// [Sample]
// User specific weather station.
FUNCTION_BLOCK FB_BA_MyWeatherStation EXTENDS FB_BA_Publisher IMPLEMENTS I_BA_MyWeatherStation
VAR_OUTPUT
	fWeatherTemperature	: REAL;
	fHumidity			: REAL;
	fBrightness			: REAL;
	
	bDisturb			: BOOL;
END_VAR
VAR
	{region 'Internal'}
		eState			: (eInit:=1, eOperation:=2, eError:=3) UDINT	:= 1;
		stData			: ST_BA_MyWeatherData;
	{endregion}
	{region 'Temporary'}
		_nCounter		: UINT;
	{endregion}
END_VAR

CASE (eState) OF
	eInit:
		IF (OnInit()) THEN
			eState := eOperation;
		ELSE
			eState := eError;
		END_IF
		
	eOperation:
		// [Sample] Simulate weather data.
		_nCounter := (_nCounter+1);
		
		IF ((_nCounter MOD 1000) > 800) THEN
			// Simulate a physical error:
			MEMSET(ADR(stData), 0, SIZEOF(stData));
			stData.fWeatherTemperature := 99.9;
			stData.fHumidity := 99.9;
			stData.bDisturb := TRUE;
		ELSE
			// Simulate valid values:
			stData.fWeatherTemperature := 20 + (TO_REAL((_nCounter / 10) MOD 100) * 0.01);
			stData.fHumidity := TO_REAL(50 + (_nCounter MOD 1000) / 500);
			stData.fBrightness := TO_REAL(10 + (_nCounter MOD 1000) / 200);
			stData.fWindSpeed := TO_REAL(5 + ((_nCounter MOD 500) / 10));
			stData.fWindDirection := TO_REAL(90 + ((_nCounter MOD 500) / 200));
			stData.fLatitude := 51.8761551;
			stData.fLongitude := 8.4671055;
			stData.bDisturb := FALSE;
		END_IF
		
END_CASE
		
// Update outputs of most important variables:
fWeatherTemperature := stData.fWeatherTemperature;
fHumidity := stData.fHumidity;
fBrightness := stData.fBrightness;
bDisturb := stData.bDisturb;

PROPERTY Brightness : REAL
GET
Brightness := stData.fBrightness;
END_GET
END_PROPERTY

PROPERTY Error : BOOL
GET
Error := (eState=eError);
END_GET
END_PROPERTY

METHOD FB_init : BOOL
VAR_INPUT
	bInitRetains : BOOL; // if TRUE, the retain variables are initialized (warm start / cold start)
	bInCopyCode : BOOL;  // if TRUE, the instance afterwards gets moved into the copy code (online change)
END_VAR
// [Hint]
// > Eigentlich wird an dieser Stelle das Profil definiert. Aber zur Übersicht wird es in "MAIN_SharedInterfaces" initialisiert.

// bEnPublish := TRUE;
// iProfile := SampleMyProfiles.MyWeatherStation;
END_METHOD

// Returns published data.
METHOD GetData
VAR_OUTPUT
	pData			: PVOID;				// Pointer to published data.
	nSize			: DINT;					// Size of published data.
END_VAR
pData := ADR(stData);
nSize := SIZEOF(stData);
END_METHOD

PROPERTY Humidity : REAL
GET
Humidity := stData.fHumidity;
END_GET
END_PROPERTY

PROPERTY Latitude : REAL
GET
Latitude := stData.fLatitude;
END_GET
END_PROPERTY

PROPERTY Longitude : REAL
GET
Longitude := stData.fLongitude;
END_GET
END_PROPERTY

METHOD PROTECTED OnInit : BOOL
IF (SUPER^.OnInit()) THEN
	// [Sample]:
	// Implement custom init code here (Optional).
	// ...
	
	OnInit := TRUE;
END_IF
END_METHOD

{attribute 'call_after_online_change_slot' := '5000'}
METHOD PROTECTED OnPostOnlineChange
SUPER^.OnPostOnlineChange();

// Re-initialize after online-changes:
eState := eInit;
END_METHOD

PROPERTY Ready : BOOL
GET
Ready := (eState=eOperation);
END_GET
END_PROPERTY

PROPERTY Valid : BOOL
GET
IF (SUPER^.Valid) THEN
	// [Sample]:
	// Implement custom validation code here (Optional).
	// ...
	
	Valid := TRUE;
END_IF
END_GET
END_PROPERTY

PROPERTY WeatherTemperature : REAL
GET
WeatherTemperature := stData.fWeatherTemperature;
END_GET
END_PROPERTY

PROPERTY WindDirection : REAL
GET
WindDirection := stData.fWindDirection;
END_GET
END_PROPERTY

PROPERTY WindSpeed : REAL
GET
WindSpeed := stData.fWindSpeed;
END_GET
END_PROPERTY

END_FUNCTION_BLOCK

(* stored: Version 1.1.0.1, ProductVersion 3.1.4024.9
   POU FB_BA_MyWeatherStation: Id {325ca01a-4181-4604-a24c-032333bda7d8}, SpecialFunc None
   Folder [Protected] Events: Id {d22c7991-1d19-4780-be08-e2352a6e2038}
   Folder Management: Id {7fe2618b-fa69-4bda-a041-90f62599a105}
   Folder Properties: Id {d11fab7a-0307-45e9-aa93-3c112e191c83}
   Folder Properties: Id {fc4a37fb-0788-49d8-868f-7f1fb6657f22}
   Property Brightness: Id {8f68b89d-f748-420d-be3c-fad39b23eceb}
   Get Get: Id {2e11ac81-73c6-4774-af98-0966db16d9b6}
   Property Error: Id {c93b8f3b-bf2e-484d-ba7f-a1ff13f92748}
   Get Get: Id {a7d3988f-c07a-4361-b40c-54447e1dc4d7}
   Method FB_init: Id {2fa2cb0a-a4b4-41de-8c4c-6d1246ad58bd}
   Method GetData: Id {a064610f-7304-45ca-afbf-43a0384c83f4}
   Property Humidity: Id {ccdd0b4e-9674-4137-b058-115e4418a811}
   Get Get: Id {206d56ad-bc2e-466a-bb11-a981ba86673d}
   Property Latitude: Id {1fa404d1-5572-4cc4-b454-c2fd6ff8db3d}
   Get Get: Id {4ae46f5c-834b-4604-beee-ebecb5b31644}
   Property Longitude: Id {30fe5788-be81-4bd4-81df-be1ca384a008}
   Get Get: Id {ecfd843e-2a59-427e-a116-b03459fc74a7}
   Method OnInit: Id {4a7b9460-4e64-426f-b877-154635ed56e3}
   Method OnPostOnlineChange: Id {8e310921-a50c-4bfc-91ac-2c44692005ae}
   Property Ready: Id {b05ad22b-ad2d-4655-8772-2b773b85e1df}
   Get Get: Id {0171a4a3-d220-4506-b7f8-59cf07047441}
   Property Valid: Id {83e6fe39-753a-453b-9b15-494d41b3fbd7}
   Get Get: Id {7a944215-4b5f-4487-99c3-d446194a8216}
   Property WeatherTemperature: Id {3e0d7e2e-264f-4754-8352-62676acf18ee}
   Get Get: Id {3e12772c-089d-4226-bfdd-12496518e9f3}
   Property WindDirection: Id {fefa4046-87ce-48b6-913f-b5193379cea0}
   Get Get: Id {279a43b1-3d6a-48a7-86f4-78e8f80fdfeb}
   Property WindSpeed: Id {e020b5b0-f346-43ad-9c0e-b7d2cc6e54e9}
   Get Get: Id {571f99b1-e9d5-46b3-8726-e8d1d983ae87} *)
